// TIA Portal V21 export
DATA_BLOCK "Dati produzione"   // DB7
{ S7_Optimized_Access := 'TRUE' }
// stored: MemoryReserve 100
   VAR RETAIN
      Misuratore : Array[0.."K_NumPortata"] of "ElencoCampionature";
      TimerCampionatura { S7_SetPoint := 'True'} : "Std_stTimer";
      CampionaturaAttuale { S7_SetPoint := 'True'} : Int := 3;
   END_VAR
   VAR
      ResetCompleto : Bool := FALSE;
   END_VAR
BEGIN
   Misuratore[0].h[1..24].OrarioCampionatura := DT#1990-01-01-00:00:00;
   Misuratore[0].h[1..24].MetriCubi := 0.0;
   TimerCampionatura.IN := TRUE;
   TimerCampionatura.O := FALSE;
   TimerCampionatura.Preset := 3600.0;
   TimerCampionatura.TempoTrascorso := 2926.036;
END_DATA_BLOCK
